FUNCTION_BLOCK TUnsupportedEventHandler IMPLEMENTS IUnsupportedEventHandler
VAR_INPUT
END_VAR
VAR_OUTPUT
END_VAR
VAR
END_VAR

END_FUNCTION_BLOCK

(* stored: Version 1.1.0.1, ProductVersion 3.1.4024.4
   POU TUnsupportedEventHandler: Id {a93b148c-62d8-436a-a14f-f2e39d309283}, SpecialFunc None *)
